ABB RobotStudio station: Entregable2.rspag

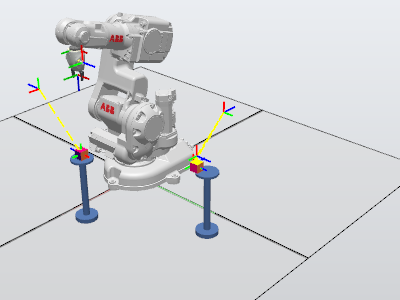
--- station ---
Station Entregable2 (saved by RobotStudio 25.2.11220.0)
Controller IRB140_6_81
  mechanical unit ROB_1: IRB140_6_81_C_03, 6 joints, base frame (0, 0, 0) mm
Layout (positions relative to the parent item):
  - IRB140_6_81_C_03 [mechanism, from %ABB.RobotStudio.Models.IRB140%\IRB140_6_81_C_G_03.rslib] at (0, 0, 0) mm; joint values [0, -0.3578, 0.0575, 0, 1.8711, 1.5708] (rad or m)
  - Smart_Gripper_Servo_One_Vacuum_Fingers [mechanism] at (306.93, 0, 736.6) mm, rotated rx -180 ry 0 rz 90 deg; joint values [0.025] (rad or m)
      TCP Servo at (0, 0, 114.2) mm
      TCP VaccumOne at (63.5, 18.5, 37.5) mm, rotated rx 0 ry 90 rz 0 deg
      links: HandBase, DownFinger, UpFinger
  - Pedestal_fijo [part] at (-400, 0, 0) mm, size 103.3 x 103.3 x 302.5 mm
  - Cubo [part] at (-400, 0, 0) mm, size 40 x 40 x 40 mm
  - Pedestal [part] at (-666.17, 471, 0) mm, size 103.3 x 103.3 x 302.5 mm
  - Cubo_2 [part] at (-162.33, 435.27, 1121.13) mm, rotated rx 0 ry 90 rz 0 deg, size 40 x 40 x 40 mm
Attachment: Smart_Gripper_Servo_One_Vacuum_Fingers is attached to IRB140_6_81_C_03 / Link6
EventTableEntry 2326: ActivationMode=2, Cyclic=false, Group=, Trigger=DO_Pinza 2327, Actions=[EventTableActionMechanicalPose 2328, EventTableActionAttach 2329], Comment=
EventTableTriggerIO 2327: Operator=0, IOValue=[1], IRC5Controller=? -1, SignalSource=IRB140_6_81 1196
EventTableActionMechanicalPose 2328: VirtualSignal=, Mechanism=Smart_Gripper_Servo_One_Vacuum_Fingers 2282, ToPoseName=Pose_cerrada, VirtualSignalValue=[1]
EventTableActionAttach 2329: MountObject=false, FlangeIndext=0, FindNearest=false, AttachmentParent=Smart_Gripper_Servo_One_Vacuum_Fingers 2282, AttachmentChild=Cubo 2307, Offset=[X=1, Y=0, Z=0, W=0, X=0, Y=1, Z=0, W=0, X=0, Y=0, Z=1, W=0, X=0, Y=0, Z=0, W=1]
EventTableTriggerIO 2381: Operator=0, IOValue=[1], IRC5Controller=? -1, SignalSource=IRB140_6_81 1196
EventTableTriggerIO 2382: Operator=0, IOValue=[1], IRC5Controller=? -1, SignalSource=IRB140_6_81 1196
EventTableTriggerIO 2383: Operator=0, IOValue=[1], IRC5Controller=? -1, SignalSource=IRB140_6_81 1196
EventTableTriggerIO 2384: Operator=0, IOValue=[1], IRC5Controller=? -1, SignalSource=IRB140_6_81 1196
EventTableTriggerIO 2399: Operator=0, IOValue=[1], IRC5Controller=? -1, SignalSource=IRB140_6_81 1196
EventTableTriggerIO 2400: Operator=0, IOValue=[1], IRC5Controller=? -1, SignalSource=IRB140_6_81 1196
EventTableTriggerIO 2401: Operator=0, IOValue=[1], IRC5Controller=? -1, SignalSource=IRB140_6_81 1196
EventTableTriggerIO 2405: Operator=0, IOValue=[1], IRC5Controller=? -1, SignalSource=IRB140_6_81 1196
EventTableTriggerIO 2406: Operator=0, IOValue=[1], IRC5Controller=? -1, SignalSource=IRB140_6_81 1196
EventTableTriggerIO 2407: Operator=0, IOValue=[1], IRC5Controller=? -1, SignalSource=IRB140_6_81 1196
EventTableTriggerIO 2408: Operator=0, IOValue=[1], IRC5Controller=? -1, SignalSource=IRB140_6_81 1196
EventTableTriggerIO 2409: Operator=0, IOValue=[1], IRC5Controller=? -1, SignalSource=IRB140_6_81 1196
EventTableTriggerIO 2436: Operator=0, IOValue=[1], IRC5Controller=? -1, SignalSource=IRB140_6_81 1196
EventTableTriggerIO 2437: Operator=0, IOValue=[1], IRC5Controller=? -1, SignalSource=IRB140_6_81 1196
EventTableTriggerIO 2438: Operator=0, IOValue=[1], IRC5Controller=? -1, SignalSource=IRB140_6_81 1196
EventTableTriggerIO 2439: Operator=0, IOValue=[1], IRC5Controller=? -1, SignalSource=IRB140_6_81 1196
EventTableTriggerIO 2440: Operator=0, IOValue=[1], IRC5Controller=? -1, SignalSource=IRB140_6_81 1196
EventTableTriggerIO 2441: Operator=0, IOValue=[1], IRC5Controller=? -1, SignalSource=IRB140_6_81 1196
EventTableTriggerIO 2442: Operator=0, IOValue=[1], IRC5Controller=? -1, SignalSource=IRB140_6_81 1196
EventTableTriggerIO 2443: Operator=0, IOValue=[1], IRC5Controller=? -1, SignalSource=IRB140_6_81 1196
EventTableTriggerIO 2444: Operator=0, IOValue=[1], IRC5Controller=? -1, SignalSource=IRB140_6_81 1196
EventTableTriggerIO 2455: Operator=0, IOValue=[1], IRC5Controller=? -1, SignalSource=IRB140_6_81 1196
EventTableTriggerIO 2456: Operator=0, IOValue=[1], IRC5Controller=? -1, SignalSource=IRB140_6_81 1196
EventTableTriggerIO 2457: Operator=0, IOValue=[1], IRC5Controller=? -1, SignalSource=IRB140_6_81 1196
EventTableTriggerIO 2458: Operator=0, IOValue=[1], IRC5Controller=? -1, SignalSource=IRB140_6_81 1196
EventTableTriggerIO 2459: Operator=0, IOValue=[1], IRC5Controller=? -1, SignalSource=IRB140_6_81 1196
EventTableTriggerIO 2460: Operator=0, IOValue=[1], IRC5Controller=? -1, SignalSource=IRB140_6_81 1196
EventTableTriggerIO 2461: Operator=0, IOValue=[1], IRC5Controller=? -1, SignalSource=IRB140_6_81 1196
EventTableTriggerIO 2462: Operator=0, IOValue=[1], IRC5Controller=? -1, SignalSource=IRB140_6_81 1196
EventTableTriggerIO 2514: Operator=0, IOValue=[1], IRC5Controller=? -1, SignalSource=IRB140_6_81 1196
EventTableTriggerIO 2516: Operator=0, IOValue=[1], IRC5Controller=? -1, SignalSource=IRB140_6_81 1196
EventTableTriggerIO 2546: Operator=0, IOValue=[1], IRC5Controller=? -1, SignalSource=IRB140_6_81 1196
EventTableTriggerIO 2547: Operator=0, IOValue=[1], IRC5Controller=? -1, SignalSource=IRB140_6_81 1196
EventTableTriggerIO 2548: Operator=0, IOValue=[1], IRC5Controller=? -1, SignalSource=IRB140_6_81 1196
EventTableTriggerIO 2549: Operator=0, IOValue=[1], IRC5Controller=? -1, SignalSource=IRB140_6_81 1196
EventTableTriggerIO 2551: Operator=0, IOValue=[1], IRC5Controller=? -1, SignalSource=IRB140_6_81 1196
EventTableTriggerIO 2553: Operator=0, IOValue=[1], IRC5Controller=? -1, SignalSource=IRB140_6_81 1196
EventTableTriggerIO 2555: Operator=0, IOValue=[1], IRC5Controller=? -1, SignalSource=IRB140_6_81 1196
EventTableTriggerIO 2556: Operator=0, IOValue=[1], IRC5Controller=? -1, SignalSource=IRB140_6_81 1196
EventTableTriggerIO 2557: Operator=0, IOValue=[1], IRC5Controller=? -1, SignalSource=IRB140_6_81 1196
EventTableTriggerIO 2558: Operator=0, IOValue=[1], IRC5Controller=? -1, SignalSource=IRB140_6_81 1196
EventTableTriggerIO 2559: Operator=0, IOValue=[1], IRC5Controller=? -1, SignalSource=IRB140_6_81 1196
EventTableTriggerIO 2560: Operator=0, IOValue=[1], IRC5Controller=? -1, SignalSource=IRB140_6_81 1196
EventTableTriggerIO 2561: Operator=0, IOValue=[1], IRC5Controller=? -1, SignalSource=IRB140_6_81 1196
EventTableTriggerIO 2562: Operator=0, IOValue=[1], IRC5Controller=? -1, SignalSource=IRB140_6_81 1196
EventTableTriggerIO 2596: Operator=0, IOValue=[1], IRC5Controller=? -1, SignalSource=IRB140_6_81 1196
EventTableTriggerIO 2597: Operator=0, IOValue=[1], IRC5Controller=? -1, SignalSource=IRB140_6_81 1196
EventTableTriggerIO 2598: Operator=0, IOValue=[1], IRC5Controller=? -1, SignalSource=IRB140_6_81 1196
EventTableTriggerIO 2605: Operator=0, IOValue=[1], IRC5Controller=? -1, SignalSource=IRB140_6_81 1196
EventTableEntry 2606: ActivationMode=2, Cyclic=false, Group=, Trigger=DO_Pinza 2607, Actions=[EventTableActionMechanicalPose 2608, EventTableActionDetach 2609], Comment=
EventTableTriggerIO 2607: Operator=0, IOValue=[0], IRC5Controller=? -1, SignalSource=IRB140_6_81 1196
EventTableActionMechanicalPose 2608: VirtualSignal=, Mechanism=Smart_Gripper_Servo_One_Vacuum_Fingers 2282, ToPoseName=Pose_abierta, VirtualSignalValue=[1]
EventTableActionDetach 2609: AttachmentParent=Smart_Gripper_Servo_One_Vacuum_Fingers 2282, AttachmentChild=Cubo 2307
EventTableTriggerIO 2610: Operator=0, IOValue=[0], IRC5Controller=? -1, SignalSource=IRB140_6_81 1196
EventTableTriggerIO 2622: Operator=0, IOValue=[1], IRC5Controller=? -1, SignalSource=IRB140_6_81 1196
EventTableTriggerIO 2623: Operator=0, IOValue=[1], IRC5Controller=? -1, SignalSource=IRB140_6_81 1196
EventTableTriggerIO 2624: Operator=0, IOValue=[1], IRC5Controller=? -1, SignalSource=IRB140_6_81 1196
EventTableTriggerIO 2625: Operator=0, IOValue=[1], IRC5Controller=? -1, SignalSource=IRB140_6_81 1196
EventTableTriggerIO 2626: Operator=0, IOValue=[1], IRC5Controller=? -1, SignalSource=IRB140_6_81 1196
EventTableTriggerIO 2627: Operator=0, IOValue=[1], IRC5Controller=? -1, SignalSource=IRB140_6_81 1196
EventTableTriggerIO 2628: Operator=0, IOValue=[1], IRC5Controller=? -1, SignalSource=IRB140_6_81 1196
EventTableTriggerIO 2629: Operator=0, IOValue=[1], IRC5Controller=? -1, SignalSource=IRB140_6_81 1196
EventTableTriggerIO 2630: Operator=0, IOValue=[1], IRC5Controller=? -1, SignalSource=IRB140_6_81 1196
EventTableTriggerIO 2631: Operator=0, IOValue=[1], IRC5Controller=? -1, SignalSource=IRB140_6_81 1196
EventTableTriggerIO 2632: Operator=0, IOValue=[1], IRC5Controller=? -1, SignalSource=IRB140_6_81 1196
EventTableTriggerIO 2633: Operator=0, IOValue=[1], IRC5Controller=? -1, SignalSource=IRB140_6_81 1196
EventTableTriggerIO 2634: Operator=0, IOValue=[1], IRC5Controller=? -1, SignalSource=IRB140_6_81 1196
EventTableTriggerIO 2635: Operator=0, IOValue=[1], IRC5Controller=? -1, SignalSource=IRB140_6_81 1196
EventTableTriggerIO 2636: Operator=0, IOValue=[1], IRC5Controller=? -1, SignalSource=IRB140_6_81 1196
EventTableTriggerIO 2637: Operator=0, IOValue=[1], IRC5Controller=? -1, SignalSource=IRB140_6_81 1196
EventTableTriggerIO 2638: Operator=0, IOValue=[1], IRC5Controller=? -1, SignalSource=IRB140_6_81 1196
EventTableTriggerIO 2639: Operator=0, IOValue=[1], IRC5Controller=? -1, SignalSource=IRB140_6_81 1196
EventTableTriggerIO 2640: Operator=0, IOValue=[1], IRC5Controller=? -1, SignalSource=IRB140_6_81 1196
EventTableTriggerIO 2641: Operator=0, IOValue=[1], IRC5Controller=? -1, SignalSource=IRB140_6_81 1196
EventTableTriggerIO 2642: Operator=0, IOValue=[0], IRC5Controller=? -1, SignalSource=IRB140_6_81 1196
EventTableTriggerIO 2643: Operator=0, IOValue=[0], IRC5Controller=? -1, SignalSource=IRB140_6_81 1196
EventTableTriggerIO 2644: Operator=0, IOValue=[0], IRC5Controller=? -1, SignalSource=IRB140_6_81 1196
EventTableTriggerIO 2645: Operator=0, IOValue=[0], IRC5Controller=? -1, SignalSource=IRB140_6_81 1196
EventTableTriggerIO 2646: Operator=0, IOValue=[0], IRC5Controller=? -1, SignalSource=IRB140_6_81 1196
EventTableTriggerIO 2647: Operator=0, IOValue=[0], IRC5Controller=? -1, SignalSource=IRB140_6_81 1196
EventTableTriggerIO 2648: Operator=0, IOValue=[0], IRC5Controller=? -1, SignalSource=IRB140_6_81 1196
EventTableTriggerIO 2649: Operator=0, IOValue=[0], IRC5Controller=? -1, SignalSource=IRB140_6_81 1196
EventTableTriggerIO 2650: Operator=0, IOValue=[0], IRC5Controller=? -1, SignalSource=IRB140_6_81 1196
EventTableTriggerIO 2651: Operator=0, IOValue=[0], IRC5Controller=? -1, SignalSource=IRB140_6_81 1196
EventTableTriggerIO 2652: Operator=0, IOValue=[0], IRC5Controller=? -1, SignalSource=IRB140_6_81 1196
EventTableTriggerIO 2653: Operator=0, IOValue=[0], IRC5Controller=? -1, SignalSource=IRB140_6_81 1196
EventTableTriggerIO 2654: Operator=0, IOValue=[0], IRC5Controller=? -1, SignalSource=IRB140_6_81 1196
EventTableTriggerIO 2655: Operator=0, IOValue=[0], IRC5Controller=? -1, SignalSource=IRB140_6_81 1196
EventTableTriggerIO 2656: Operator=0, IOValue=[0], IRC5Controller=? -1, SignalSource=IRB140_6_81 1196
EventTableTriggerIO 2657: Operator=0, IOValue=[0], IRC5Controller=? -1, SignalSource=IRB140_6_81 1196
EventTableTriggerIO 2658: Operator=0, IOValue=[0], IRC5Controller=? -1, SignalSource=IRB140_6_81 1196
EventTableTriggerIO 2659: Operator=0, IOValue=[0], IRC5Controller=? -1, SignalSource=IRB140_6_81 1196
EventTableTriggerIO 2660: Operator=0, IOValue=[0], IRC5Controller=? -1, SignalSource=IRB140_6_81 1196
EventTableTriggerIO 2661: Operator=0, IOValue=[0], IRC5Controller=? -1, SignalSource=IRB140_6_81 1196
EventTableEntry 2662: ActivationMode=2, Cyclic=false, Group=, Trigger=DO_Vacum 2663, Actions=[EventTableActionAttach 2664], Comment=
EventTableTriggerIO 2663: Operator=0, IOValue=[1], IRC5Controller=? -1, SignalSource=IRB140_6_81 1196
EventTableActionAttach 2664: MountObject=false, FlangeIndext=0, FindNearest=false, AttachmentParent=Smart_Gripper_Servo_One_Vacuum_Fingers 2282, AttachmentChild=Cubo_2 2621, Offset=[X=1, Y=0, Z=0, W=0, X=0, Y=1, Z=0, W=0, X=0, Y=0, Z=1, W=0, X=0, Y=0, Z=0, W=1]
EventTableTriggerIO 2665: Operator=0, IOValue=[1], IRC5Controller=? -1, SignalSource=IRB140_6_81 1196
EventTableTriggerIO 2666: Operator=0, IOValue=[1], IRC5Controller=? -1, SignalSource=IRB140_6_81 1196
EventTableTriggerIO 2667: Operator=0, IOValue=[1], IRC5Controller=? -1, SignalSource=IRB140_6_81 1196
EventTableTriggerIO 2668: Operator=0, IOValue=[1], IRC5Controller=? -1, SignalSource=IRB140_6_81 1196
EventTableTriggerIO 2669: Operator=0, IOValue=[1], IRC5Controller=? -1, SignalSource=IRB140_6_81 1196
EventTableTriggerIO 2670: Operator=0, IOValue=[1], IRC5Controller=? -1, SignalSource=IRB140_6_81 1196
EventTableTriggerIO 2671: Operator=0, IOValue=[1], IRC5Controller=? -1, SignalSource=IRB140_6_81 1196
EventTableTriggerIO 2672: Operator=0, IOValue=[1], IRC5Controller=? -1, SignalSource=IRB140_6_81 1196
EventTableTriggerIO 2673: Operator=0, IOValue=[1], IRC5Controller=? -1, SignalSource=IRB140_6_81 1196
EventTableTriggerIO 2674: Operator=0, IOValue=[1], IRC5Controller=? -1, SignalSource=IRB140_6_81 1196
EventTableTriggerIO 2675: Operator=0, IOValue=[1], IRC5Controller=? -1, SignalSource=IRB140_6_81 1196
EventTableTriggerIO 2676: Operator=0, IOValue=[1], IRC5Controller=? -1, SignalSource=IRB140_6_81 1196
EventTableTriggerIO 2677: Operator=0, IOValue=[1], IRC5Controller=? -1, SignalSource=IRB140_6_81 1196
EventTableTriggerIO 2678: Operator=0, IOValue=[1], IRC5Controller=? -1, SignalSource=IRB140_6_81 1196
EventTableTriggerIO 2679: Operator=0, IOValue=[1], IRC5Controller=? -1, SignalSource=IRB140_6_81 1196
EventTableTriggerIO 2680: Operator=0, IOValue=[1], IRC5Controller=? -1, SignalSource=IRB140_6_81 1196
EventTableTriggerIO 2681: Operator=0, IOValue=[1], IRC5Controller=? -1, SignalSource=IRB140_6_81 1196
EventTableTriggerIO 2682: Operator=0, IOValue=[1], IRC5Controller=? -1, SignalSource=IRB140_6_81 1196
EventTableTriggerIO 2683: Operator=0, IOValue=[1], IRC5Controller=? -1, SignalSource=IRB140_6_81 1196
EventTableTriggerIO 2684: Operator=0, IOValue=[1], IRC5Controller=? -1, SignalSource=IRB140_6_81 1196
EventTableEntry 2685: ActivationMode=2, Cyclic=false, Group=, Trigger=DO_Vacum 2686, Actions=[EventTableActionDetach 2687], Comment=
EventTableTriggerIO 2686: Operator=0, IOValue=[0], IRC5Controller=? -1, SignalSource=IRB140_6_81 1196
EventTableActionDetach 2687: AttachmentParent=Smart_Gripper_Servo_One_Vacuum_Fingers 2282, AttachmentChild=Cubo_2 2621
EventTableTriggerIO 2688: Operator=0, IOValue=[0], IRC5Controller=? -1, SignalSource=IRB140_6_81 1196
EventTableTriggerIO 2689: Operator=0, IOValue=[0], IRC5Controller=? -1, SignalSource=IRB140_6_81 1196
EventTableTriggerIO 2690: Operator=0, IOValue=[0], IRC5Controller=? -1, SignalSource=IRB140_6_81 1196
EventTableTriggerIO 2691: Operator=0, IOValue=[0], IRC5Controller=? -1, SignalSource=IRB140_6_81 1196
EventTableTriggerIO 2692: Operator=0, IOValue=[0], IRC5Controller=? -1, SignalSource=IRB140_6_81 1196
EventTableTriggerIO 2693: Operator=0, IOValue=[0], IRC5Controller=? -1, SignalSource=IRB140_6_81 1196
EventTableTriggerIO 2694: Operator=0, IOValue=[0], IRC5Controller=? -1, SignalSource=IRB140_6_81 1196
EventTableTriggerIO 2695: Operator=0, IOValue=[0], IRC5Controller=? -1, SignalSource=IRB140_6_81 1196
EventTableTriggerIO 2696: Operator=0, IOValue=[0], IRC5Controller=? -1, SignalSource=IRB140_6_81 1196
EventTableTriggerIO 2697: Operator=0, IOValue=[0], IRC5Controller=? -1, SignalSource=IRB140_6_81 1196
EventTableTriggerIO 2698: Operator=0, IOValue=[0], IRC5Controller=? -1, SignalSource=IRB140_6_81 1196
EventTableTriggerIO 2699: Operator=0, IOValue=[0], IRC5Controller=? -1, SignalSource=IRB140_6_81 1196
EventTableTriggerIO 2700: Operator=0, IOValue=[0], IRC5Controller=? -1, SignalSource=IRB140_6_81 1196
EventTableTriggerIO 2701: Operator=0, IOValue=[0], IRC5Controller=? -1, SignalSource=IRB140_6_81 1196
EventTableTriggerIO 2702: Operator=0, IOValue=[0], IRC5Controller=? -1, SignalSource=IRB140_6_81 1196
EventTableTriggerIO 2703: Operator=0, IOValue=[0], IRC5Controller=? -1, SignalSource=IRB140_6_81 1196
EventTableTriggerIO 2704: Operator=0, IOValue=[0], IRC5Controller=? -1, SignalSource=IRB140_6_81 1196
EventTableTriggerIO 2705: Operator=0, IOValue=[0], IRC5Controller=? -1, SignalSource=IRB140_6_81 1196
EventTableTriggerIO 2706: Operator=0, IOValue=[0], IRC5Controller=? -1, SignalSource=IRB140_6_81 1196
EventTableTriggerIO 2707: Operator=0, IOValue=[0], IRC5Controller=? -1, SignalSource=IRB140_6_81 1196
EventTableTriggerIO 2804: Operator=0, IOValue=[1], IRC5Controller=? -1, SignalSource=IRB140_6_81 1196
EventTableTriggerIO 2805: Operator=0, IOValue=[1], IRC5Controller=? -1, SignalSource=IRB140_6_81 1196
EventTableTriggerIO 2806: Operator=0, IOValue=[0], IRC5Controller=? -1, SignalSource=IRB140_6_81 1196
EventTableTriggerIO 2807: Operator=0, IOValue=[0], IRC5Controller=? -1, SignalSource=IRB140_6_81 1196
EventTableTriggerIO 2808: Operator=0, IOValue=[1], IRC5Controller=? -1, SignalSource=IRB140_6_81 1196
EventTableTriggerIO 2809: Operator=0, IOValue=[1], IRC5Controller=? -1, SignalSource=IRB140_6_81 1196
EventTableTriggerIO 2810: Operator=0, IOValue=[0], IRC5Controller=? -1, SignalSource=IRB140_6_81 1196
EventTableTriggerIO 2811: Operator=0, IOValue=[0], IRC5Controller=? -1, SignalSource=IRB140_6_81 1196
EventTableTriggerIO 2812: Operator=0, IOValue=[1], IRC5Controller=? -1, SignalSource=IRB140_6_81 1196
EventTableTriggerIO 2813: Operator=0, IOValue=[1], IRC5Controller=? -1, SignalSource=IRB140_6_81 1196
EventTableTriggerIO 2814: Operator=0, IOValue=[1], IRC5Controller=? -1, SignalSource=IRB140_6_81 1196
EventTableTriggerIO 2815: Operator=0, IOValue=[1], IRC5Controller=? -1, SignalSource=IRB140_6_81 1196
EventTableTriggerIO 2816: Operator=0, IOValue=[0], IRC5Controller=? -1, SignalSource=IRB140_6_81 1196
EventTableTriggerIO 2817: Operator=0, IOValue=[0], IRC5Controller=? -1, SignalSource=IRB140_6_81 1196
EventTableTriggerIO 2818: Operator=0, IOValue=[0], IRC5Controller=? -1, SignalSource=IRB140_6_81 1196
EventTableTriggerIO 2819: Operator=0, IOValue=[0], IRC5Controller=? -1, SignalSource=IRB140_6_81 1196
EventTableTriggerIO 2820: Operator=0, IOValue=[1], IRC5Controller=? -1, SignalSource=IRB140_6_81 1196
EventTableTriggerIO 2821: Operator=0, IOValue=[1], IRC5Controller=? -1, SignalSource=IRB140_6_81 1196
EventTableTriggerIO 2822: Operator=0, IOValue=[1], IRC5Controller=? -1, SignalSource=IRB140_6_81 1196
EventTableTriggerIO 2823: Operator=0, IOValue=[1], IRC5Controller=? -1, SignalSource=IRB140_6_81 1196
EventTableTriggerIO 2824: Operator=0, IOValue=[0], IRC5Controller=? -1, SignalSource=IRB140_6_81 1196
EventTableTriggerIO 2825: Operator=0, IOValue=[0], IRC5Controller=? -1, SignalSource=IRB140_6_81 1196
EventTableTriggerIO 2826: Operator=0, IOValue=[0], IRC5Controller=? -1, SignalSource=IRB140_6_81 1196
EventTableTriggerIO 2827: Operator=0, IOValue=[0], IRC5Controller=? -1, SignalSource=IRB140_6_81 1196
Targets, tools, work objects and paths stored in the station and not in the controller backup, written as RAPID:
! task T_ROB1
MODULE Module1
  CONST robtarget giro_y_90:=[[506.933,0,622.4],[0.707106781,0.707106781,0,0],[-2,1,-2,6],[9E+09,9E+09,9E+09,9E+09,9E+09,9E+09]];
  CONST robtarget Posicion_final_1:=[[400,100,320],[0.707106781,0.707106781,0,0],[0,-1,-2,0],[9E+09,9E+09,9E+09,9E+09,9E+09,9E+09]];
  CONST robtarget Posicion_coger_2:=[[157.667,515.273,321.132],[0.5,-0.5,-0.5,-0.5],[0,0,0,0],[9E+09,9E+09,9E+09,9E+09,9E+09,9E+09]];
  CONST robtarget Home_2:=[[325.433,63.5,699.1],[0.5,-0.5,-0.5,-0.5],[-1,0,0,0],[9E+09,9E+09,9E+09,9E+09,9E+09,9E+09]];
  CONST robtarget Posicion_final_2:=[[157.667,515.273,321.132],[0.707106781,0,-0.707106781,0],[0,0,0,0],[9E+09,9E+09,9E+09,9E+09,9E+09,9E+09]];
  CONST robtarget Punto_help:=[[157.667,535.273,368.720557964],[0.5,-0.5,-0.5,-0.5],[0,0,0,0],[9E+09,9E+09,9E+09,9E+09,9E+09,9E+09]];
  CONST robtarget giro_x_90:=[[-62.615343749,490.552913165,472.156538127],[0.707106781,0,-0.707106781,0],[0,0,0,0],[9E+09,9E+09,9E+09,9E+09,9E+09,9E+09]];
  PROC Gripper()
    MoveL Posicion_coger,v1000,z100,Servo\WObj:=wobj0;
    WaitTime 2;
    SetDO DO_Pinza,1;
    MoveJ giro_y_90,v200,fine,Servo\WObj:=wobj0;
    MoveJ Posicion_final_1,v200,fine,Servo\WObj:=wobj0;
    WaitTime 2;
    Reset DO_Pinza;
  ENDPROC
  PROC Vaccum()
    MoveL Posicion_coger_2,v200,fine,VaccumOne\WObj:=wobj0;
    WaitTime 2;
    SetDO DO_Vacum,1;
    MoveL Punto_help,v200,fine,VaccumOne\WObj:=wobj0;
    MoveJ giro_x_90,v200,fine,VaccumOne\WObj:=wobj0;
    MoveJ Posicion_final_2,v200,fine,VaccumOne\WObj:=wobj0;
    WaitTime 2;
    Reset DO_Pinza;
  ENDPROC
ENDMODULE


--- Controller Data/IRB140_6_81/RAPID/TASK1/PROGMOD/CalibData.mod ---
MODULE CalibData
    PERS tooldata Servo:=[TRUE,[[0,0,114.2],[1,0,0,0]],[0.226,[8.9,12.3,48.7],[1,0,0,0],0.00021,0.00024,0.00009]];
    PERS tooldata VaccumOne:=[TRUE,[[63.5,18.5,37.5],[0.707107,0,0.707107,0]],[0.226,[8.9,12.3,48.7],[1,0,0,0],0.00021,0.00024,9E-5]];
ENDMODULE

--- Controller Data/IRB140_6_81/RAPID/TASK1/PROGMOD/Module1.mod ---
MODULE Module1
    CONST robtarget Home:=[[306.933,0,622.4],[1,0,0,0],[0,0,0,0],[9E+09,9E+09,9E+09,9E+09,9E+09,9E+09]];
    CONST robtarget Posicion_coger:=[[400,100,340],[0,0.707106781,0.707106781,0],[0,0,1,0],[9E+09,9E+09,9E+09,9E+09,9E+09,9E+09]];
    TASK PERS wobjdata wobj1:=[FALSE,TRUE,"",[[0,0,0],[1,0,0,0]],[[0,0,0],[1,0,0,0]]];
    !***********************************************************
    !
    ! M?dulo:  Module1
    !
    ! Descripción:
    !   <Introduzca la descripción aquí>
    !
    ! Autor: r.castilla.2023
    !
    ! Versión: 1.0
    !
    !***********************************************************


    !***********************************************************
    !
    ! Procedimiento Main
    !
    !   Este es el punto de entrada de su programa
    !
    !***********************************************************
    PROC main()
        !Add your code here
    ENDPROC
    PROC Path_10()
        MoveL Home,v1000,z100,Servo\WObj:=wobj0;
        MoveL Posicion_coger,v1000,z100,Servo\WObj:=wobj0;
        SetDO DO_Pinza,1;
        WaitTime 2;
        MoveL Home,v1000,z100,Servo\WObj:=wobj0;
    ENDPROC
ENDMODULE

--- Controller Data/IRB140_6_81/SYSPAR/EIO.cfg ---
EIO:CFG_1.0:6:1::
#
EIO_SIGNAL:

      -Name "DO_Pinza" -SignalType "DO" -Access "All"

      -Name "DO_Vacum" -SignalType "DO" -Access "All"
